// Mitsubishi GX Works2 project: a4   PLC: Q02/Q02H

PROGRAM MAIN
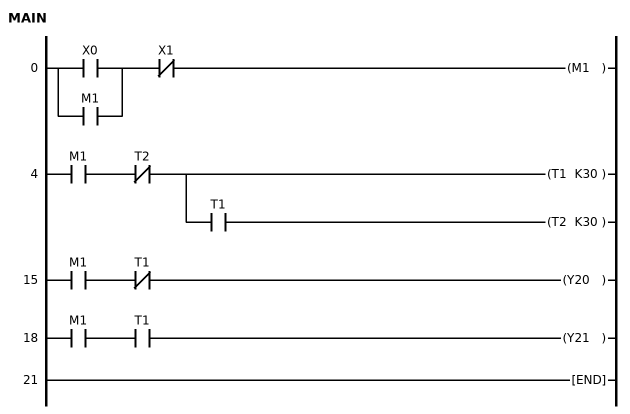
0     LD      X0
      OR      M1
      ANI     X1
      OUT     M1
4     LD      M1
      ANI     T2
      OUT     T1 K30
      AND     T1
      OUT     T2 K30
15    LD      M1
      ANI     T1
      OUT     Y20
18    LD      M1
      AND     T1
      OUT     Y21
21    END
END_PROGRAM
